// TIA Portal V17 export
// export: Created 2025-03-05T08:02:08.4539629Z, ExportSetting WithDefaults, DisplayName Totally Integrated Automation Portal, DisplayVersion V17 Update 8, DisplayName TIA Portal Openness, DisplayVersion V17 Update 8, DisplayName TIA Portal Version Control Interface, DisplayVersion V17, DisplayName SINAMICS Startdrive Advanced, DisplayVersion V17 SP2, DisplayName SINAMICS Startdrive G110M, G120, G120C, G120D, G120P, G115D, DisplayVersion V17 SP2, DisplayName SINAMICS Startdrive G130, G150, S120, S150, SINAMICS MV, S210, DisplayVersion V17 SP2, DisplayName STEP 7 Professional, DisplayVersion V17 Update 8, DisplayName SINUMERIK ONE STEP 7 Toolbox, DisplayVersion V17 Update 12, DisplayName SINUMERIK 840D sl STEP 7 Toolbox, DisplayVersion V17 Update 12, DisplayName STEP 7 Safety, DisplayVersion V17 Update 6, DisplayName WinCC Advanced, DisplayVersion V17 Update 8
TYPE "SPINDLE"
// stored: IsFailsafeCompliant false
   STRUCT
      SELECTED { ExternalVisible := 'False'; ExternalWritable := 'False'} : Bool;   // SELECTED
      CONT_INCRMTL_MODE { ExternalVisible := 'False'; ExternalWritable := 'False'} : Bool;   // CONTINOUS INCRMTL MODE
      HMI_JOG_MINUS_RQ { ExternalVisible := 'False'; ExternalWritable := 'False'} : Bool;   // HMI JOG MINUS REQUEST
      HMI_JOG_PLUS_RQ { ExternalVisible := 'False'; ExternalWritable := 'False'} : Bool;   // HMI JOG PLUS REQUEST
      HMI_JOG_MINUS_CMM { ExternalVisible := 'False'; ExternalWritable := 'False'} : Bool;   // HMI JOG MINUS COMMAND
      HMI_JOG_PLUS_CMM { ExternalVisible := 'False'; ExternalWritable := 'False'} : Bool;   // HMI JOG PLUS COMMAND
      SPEED_REACHED { ExternalVisible := 'False'; ExternalWritable := 'False'} : Bool;   // SPEED REACHED
      SPEED_ZERO { ExternalVisible := 'False'; ExternalWritable := 'False'} : Bool;   // SPEED ZERO
      JOG_HELP { ExternalVisible := 'False'; ExternalWritable := 'False'} : Bool;   // JOG HELP
      MINUS_BUTTON_HELP { ExternalVisible := 'False'; ExternalWritable := 'False'} : Bool;   // MINUS BUTTON HELP
      PLUS_BUTTON_HELP { ExternalVisible := 'False'; ExternalWritable := 'False'} : Bool;   // PLUS BUTTON HELP
      OPERATOR_HELP { ExternalVisible := 'False'; ExternalWritable := 'False'} : Bool;   // OPERATOR HELP
   END_STRUCT;
END_TYPE
